FUNCTION_BLOCK AIO_IN (* Service Interface Function Block Type *)
  (* Standard: 61499-2 *)
  (* Version 0.0, 19/05/2021, josef, nxtControl GmBH, template *)
  PACKAGE Flexbridge.Iceblock;
  (* Compiler Cpp nxtControl builtin 1.0 *)
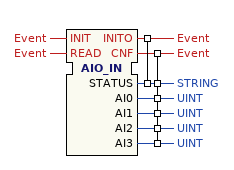
  EVENT_INPUT
    INIT;
    READ;
  END_EVENT
  EVENT_OUTPUT
    INITO WITH STATUS;
    CNF WITH STATUS, AI0, AI1, AI2, AI3;
  END_EVENT
  VAR_OUTPUT
    STATUS : STRING; (* Service Status *)
    AI0 : UINT;
    AI1 : UINT;
    AI2 : UINT;
    AI3 : UINT;
  END_VAR
  SERVICE AIO_IN/RESOURCE
    SEQUENCE normal_establishment
      AIO_IN.INIT+(PARAMS) -> RESOURCE.initialize(PARAMS) -> AIO_IN.INITO+();
    END_SEQUENCE
    SEQUENCE unsuccessful_establishment
      AIO_IN.INIT+(PARAMS) -> RESOURCE.initialize(PARAMS) -> AIO_IN.INITO-(STATUS);
    END_SEQUENCE
    SEQUENCE request_confirm
      AIO_IN.REQ+(SD) -> RESOURCE.request(SD) -> AIO_IN.CNF+(RD);
    END_SEQUENCE
    SEQUENCE request_inhibited
      AIO_IN.REQ-(SD) -> AIO_IN.CNF-(STATUS);
    END_SEQUENCE
    SEQUENCE request_error
      AIO_IN.REQ+(SD) -> RESOURCE.request(SD) -> AIO_IN.CNF-(STATUS);
    END_SEQUENCE
    SEQUENCE indication_response
      RESOURCE.indicate(RD) -> AIO_IN.IND+(RD);
      AIO_IN.RSP(QI,SD) -> RESOURCE.response(QI,SD);
    END_SEQUENCE
    SEQUENCE indication_inhibited
      RESOURCE.indicate(RD,QI=FALSE) -> RESOURCE.inhibited();
    END_SEQUENCE
    SEQUENCE error_indication
      RESOURCE.error(STATUS) -> AIO_IN.IND-(STATUS);
    END_SEQUENCE
    SEQUENCE application_initiated_termination
      AIO_IN.INIT-() -> RESOURCE.terminate() -> AIO_IN.INITO-(STATUS);
    END_SEQUENCE
    SEQUENCE resource_initiated_termination
      -> AIO_IN.INITO-(STATUS);
    END_SEQUENCE
  END_SERVICE
END_FUNCTION_BLOCK
